(* Logix 5000 project; controller Ceca_1650T_Press 5069-L306ERM rev 32.12; software revision 32.02; part 3 of 3 *)
(* tags used below, declared in another part *)
   AUTO_CYCLE_ENABLED : BOOL;   // M0014 HMI SELECTION
   AUTO_CYCLE_SELECTED : BOOL;   // HMI BUTTON/SELECTION B0102
   AUTO_CYCLE_STOP_PB : BOOL;   // B0024
   AUTO_ONE_CYCLE_ENABLED : BOOL;   // M0013 HMI SELECTION
   AUTO_ONE_CYCLE_SELECTED : BOOL;   // HMI BUTTON/SELECTION B0101
   AUTO_UPPER_ASSIST : BOOL;   // ENCODER SIGNAL B0152
   AUTO_UPPER_ASSIST_POSITION_MINUS : REAL;
   AUTO_UPPER_ASSIST_POSITION_PLUS : REAL;
   AUTO_UPPER_LIMIT : BOOL;   // ENCODER SIGNAL B0151
   AUTO_UPPER_LIMIT_POSITION_MINUS : REAL;
   AUTO_UPPER_LIMIT_POSITION_PLUS : REAL;
   BLANKING_OFF_SIGNAL : TIMER;   // T0018
   BLANKING_PS_ENABLED : BOOL;   // M0018
   BOLSTER_DISABLED : BOOL;   // M0010
   CYCLE_STOP : BOOL;   // M0246
   DIE_CHANGE_ENABLED : BOOL;   // M0015
   DIE_CHANGE_MODE : BOOL;   // HMI BUTTON/SELECTION B0103
   DIE_SET_CHANGING : BOOL;   // B0037
   DIE_SET_CYLINDER_IN_PB : BOOL;   // B0076
   DIE_SET_CYLINDER_OUT : BOOL;   // M0217
   DIE_SET_CYLINDER_OUT_PB : BOOL;   // B0077
   DRAW_UP_ASSIST : BOOL;   // M007C
   FILTER_CLOGGED_FAULT : BOOL;   // M0023
   FRONT_SUTTER_ON_LIMIT : BOOL;   // B000C
   HMI_START_PUMPS : BOOL;   // HMI BUTTON
   INCH_ENABLED : BOOL;   // M0012 HMI SELECTION
   INCHING_SELECTED : BOOL;   // HMI BUTTON/SELECTION B0100
   Job_Call_Recipe : Recipe_Setup[50];
   L_DIECUSHION_AUTO_UP_ASSIST : BOOL;   // ENCODER SIGNAL B015A
   L_DIECUSHION_AUTO_UP_LIMIT : BOOL;   // B0156 ENCODER SIGNAL
   load_PB : BOOL;
   LOCKING_OFF_ASSIST : BOOL;   // M0032
   LUBE_LEVEL_FAULT : BOOL;   // M0022
   Machine_Current_Job : DINT;
   MAIN_PRESS_DOWN : BOOL;   // M0045
   MAIN_PRESS_POSITION_SICK : REAL;
   MAIN_PRESS_SLOW_DOWN : BOOL;   // M0046
   MAIN_PRESS_SLOW_UP : BOOL;   // M0042
   MAIN_PRESS_UP : BOOL;   // M0041
   MAIN_UPPER_LIMIT : BOOL;   // B0000
   OIL_COOLER_START : BOOL;   // B0144
   OIL_TEMP_TOO_HIGH : BOOL;   // B0143
   OIL_TEMP_WARM_UP_ON_SELECT : BOOL;   // B002C HMI BUTTON
   OIL_TEMP_WARM_UP_START : BOOL;   // B0038
   OIL_TEMPERATURE_FAULT : BOOL;   // M0025
   OIL_WORKING_LEVEL_FAULT : BOOL;   // M0021
   OPERATION_ON : BOOL;   // B0020
   PILOT_CHECK_OPEN_VALVE : BOOL;   // B0048
   PILOT_PUMP_HIGH_PRESSURE_VALVE : BOOL;   // B0060
   PILOT_PUMP_MIDDLE_PRESSURE_VALVE : BOOL;   // B0062
   PILOT_PUMP_ON : BOOL;   // B002E
   PRESS_AUTO_RUN : BOOL;   // M0069
   PRESS_HAS_A_FAULT : BOOL;   // M0027
   PRESS_HAS_A_FAULT_2 : BOOL;   // M0028
   PUMP_RUN : BOOL;   // B0021
   PUMP_START : BOOL;   // B1000
   PUMP_STOP_SIGNAL : BOOL;   // B0030
   R_DIECUSHION_AUTO_UP_ASSIST : BOOL;   // B015B ENCODER SIGNAL
   R_DIECUSHION_AUTO_UP_LIMIT : BOOL;   // B0158 ENCODER SIGNAL
   REAR_SHUTTER_ON_LIMIT : BOOL;   // B000D
   Recipe_Max : DINT;
   Recipe_Name_Pointer : DINT;
   Recipe_Number : COUNTER;
   Save_Delay : TIMER;
   save_pb : BOOL;
   Scroll_Down : BOOL;
   Scroll_up : BOOL;
   SickAFxWS_Enc1_AOI : SICK_AFX60_A101WS_A103WS_AOI;
   SickAFxWS_Enc1_Cyclic_GetSet : BOOL;
   SickAFxWS_Enc1_Init_GetSet : BOOL;
   SickAFxWS_Enc1_Timer_GetSet : TIMER;
   SLIDE_SLOW_DOWN_SIGNAL : BOOL;   // B0154 ENCODER SIGNAL
   SLIDE_SLOW_DOWN_SIGNAL_POSITION_MINUS : REAL;
   SLIDE_SLOW_DOWN_SIGNAL_POSITION_PLUS : REAL;
   TRM1 : BOOL;   // B1003
   TRM1_TIMER : TIMER;   // 5 SECONDS
   TRM2 : BOOL;   // B1001
   TRM2_TIMER : TIMER;   // 5 SECONDS
   TRM3 : BOOL;   // B1002
   TRM3_TIMER : TIMER;   // 1 SECOND
   WARM_UP_FINISHED : BOOL;   // M009E
   WARM_UP_OFF_TEMP : BOOL;   // B0027
   WARM_UP_ON : BOOL;   // M009D
   WARM_UP_ON_TIMING : TIMER;   // T0023
   WARM_UP_SELECT_OFF_TIMER : TIMER;   // T0024
   WARM_UP_SELECT_ON_TIMER : TIMER;   // T0025
(* MainProgram, continued *)

ROUTINE Modes   (* ladder *)
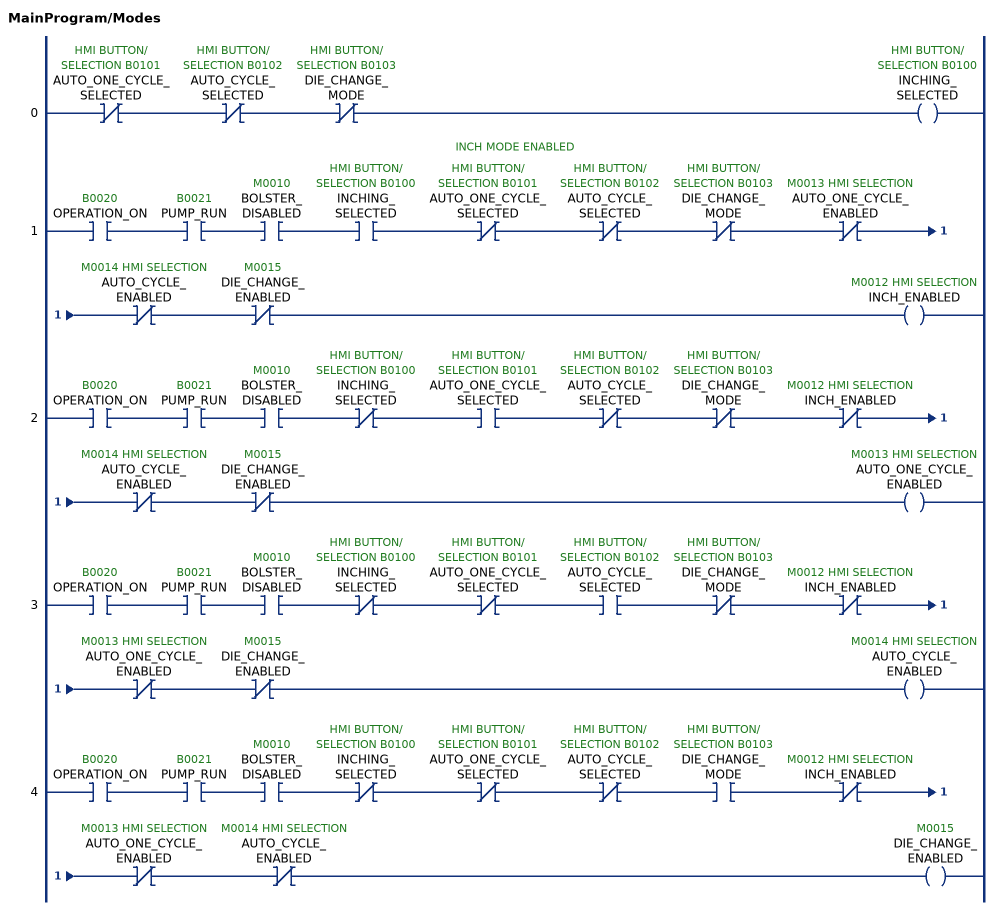
   0: XIO(AUTO_ONE_CYCLE_SELECTED)XIO(AUTO_CYCLE_SELECTED)XIO(DIE_CHANGE_MODE)OTE(INCHING_SELECTED);
   // INCH MODE ENABLED
   1: XIC(OPERATION_ON)XIC(PUMP_RUN)XIC(BOLSTER_DISABLED)XIC(INCHING_SELECTED)XIO(AUTO_ONE_CYCLE_SELECTED)XIO(AUTO_CYCLE_SELECTED)XIO(DIE_CHANGE_MODE)XIO(AUTO_ONE_CYCLE_ENABLED)XIO(AUTO_CYCLE_ENABLED)XIO(DIE_CHANGE_ENABLED)OTE(INCH_ENABLED);
   2: XIC(OPERATION_ON)XIC(PUMP_RUN)XIC(BOLSTER_DISABLED)XIO(INCHING_SELECTED)XIC(AUTO_ONE_CYCLE_SELECTED)XIO(AUTO_CYCLE_SELECTED)XIO(DIE_CHANGE_MODE)XIO(INCH_ENABLED)XIO(AUTO_CYCLE_ENABLED)XIO(DIE_CHANGE_ENABLED)OTE(AUTO_ONE_CYCLE_ENABLED);
   3: XIC(OPERATION_ON)XIC(PUMP_RUN)XIC(BOLSTER_DISABLED)XIO(INCHING_SELECTED)XIO(AUTO_ONE_CYCLE_SELECTED)XIC(AUTO_CYCLE_SELECTED)XIO(DIE_CHANGE_MODE)XIO(INCH_ENABLED)XIO(AUTO_ONE_CYCLE_ENABLED)XIO(DIE_CHANGE_ENABLED)OTE(AUTO_CYCLE_ENABLED);
   4: XIC(OPERATION_ON)XIC(PUMP_RUN)XIC(BOLSTER_DISABLED)XIO(INCHING_SELECTED)XIO(AUTO_ONE_CYCLE_SELECTED)XIO(AUTO_CYCLE_SELECTED)XIC(DIE_CHANGE_MODE)XIO(INCH_ENABLED)XIO(AUTO_ONE_CYCLE_ENABLED)XIO(AUTO_CYCLE_ENABLED)OTE(DIE_CHANGE_ENABLED);
END_ROUTINE

ROUTINE Outputs   (* ladder *)
END_ROUTINE

ROUTINE Pilot_Pump   (* ladder *)
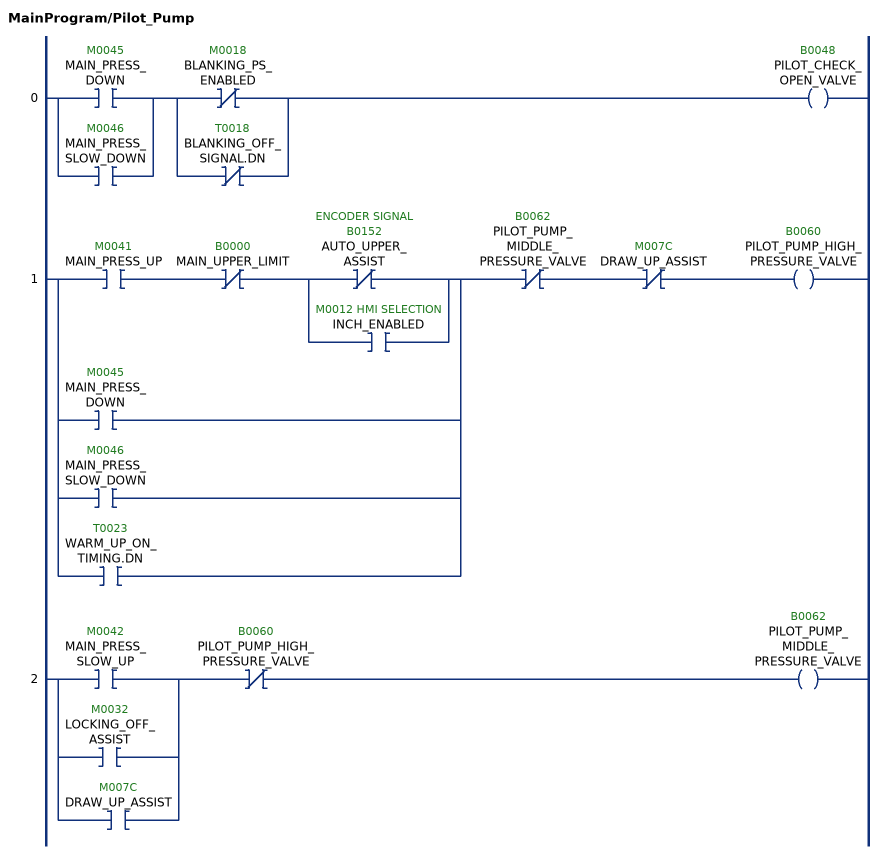
   0: [XIC(MAIN_PRESS_DOWN) ,XIC(MAIN_PRESS_SLOW_DOWN) ][XIO(BLANKING_PS_ENABLED) ,XIO(BLANKING_OFF_SIGNAL.DN) ]OTE(PILOT_CHECK_OPEN_VALVE);
   1: [XIC(MAIN_PRESS_UP) XIO(MAIN_UPPER_LIMIT) [XIO(AUTO_UPPER_ASSIST) ,XIC(INCH_ENABLED) ] ,XIC(MAIN_PRESS_DOWN) ,XIC(MAIN_PRESS_SLOW_DOWN) ,XIC(WARM_UP_ON_TIMING.DN) ]XIO(PILOT_PUMP_MIDDLE_PRESSURE_VALVE)XIO(DRAW_UP_ASSIST)OTE(PILOT_PUMP_HIGH_PRESSURE_VALVE);
   2: [XIC(MAIN_PRESS_SLOW_UP) ,XIC(LOCKING_OFF_ASSIST) ,XIC(DRAW_UP_ASSIST) ]XIO(PILOT_PUMP_HIGH_PRESSURE_VALVE)OTE(PILOT_PUMP_MIDDLE_PRESSURE_VALVE);
END_ROUTINE

ROUTINE Recipe   (* ladder *)
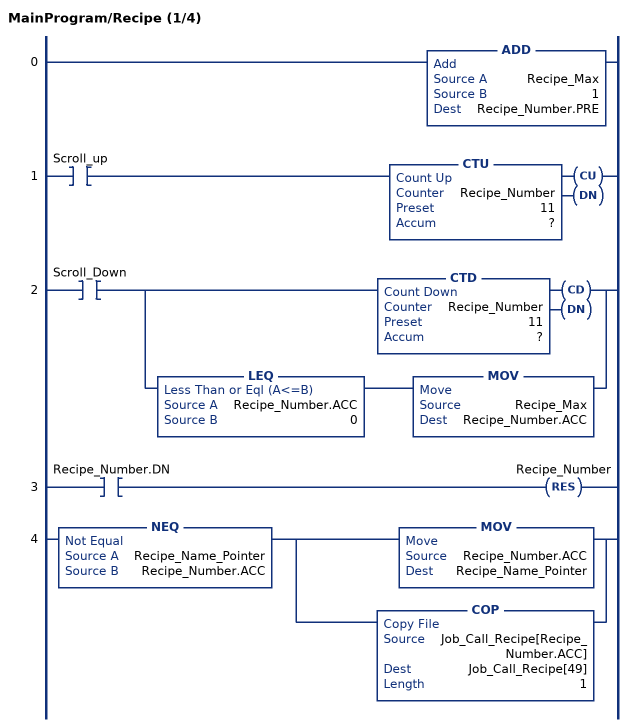
   0: ADD(Recipe_Max,1,Recipe_Number.PRE);
   1: XIC(Scroll_up)CTU(Recipe_Number,?,?);
   2: XIC(Scroll_Down)[CTD(Recipe_Number,?,?) ,LEQ(Recipe_Number.ACC,0) MOV(Recipe_Max,Recipe_Number.ACC) ];
   3: XIC(Recipe_Number.DN)RES(Recipe_Number);
   4: NEQ(Recipe_Name_Pointer,Recipe_Number.ACC)[MOV(Recipe_Number.ACC,Recipe_Name_Pointer) ,COP(Job_Call_Recipe[Recipe_Number.ACC],Job_Call_Recipe[49],1) ];
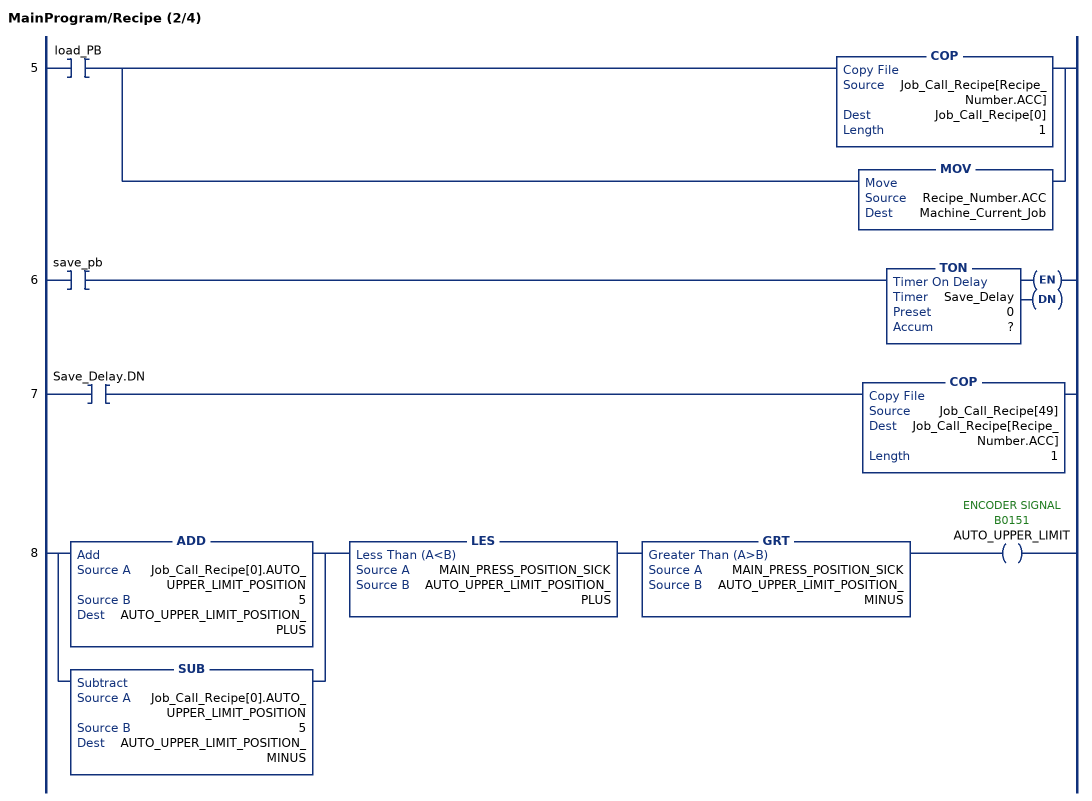
   5: XIC(load_PB)[COP(Job_Call_Recipe[Recipe_Number.ACC],Job_Call_Recipe[0],1) ,MOV(Recipe_Number.ACC,Machine_Current_Job) ];
   6: XIC(save_pb)TON(Save_Delay,?,?);
   7: XIC(Save_Delay.DN)COP(Job_Call_Recipe[49],Job_Call_Recipe[Recipe_Number.ACC],1);
   8: [ADD(Job_Call_Recipe[0].AUTO_UPPER_LIMIT_POSITION,5,AUTO_UPPER_LIMIT_POSITION_PLUS) ,SUB(Job_Call_Recipe[0].AUTO_UPPER_LIMIT_POSITION,5,AUTO_UPPER_LIMIT_POSITION_MINUS) ]LES(MAIN_PRESS_POSITION_SICK,AUTO_UPPER_LIMIT_POSITION_PLUS)GRT(MAIN_PRESS_POSITION_SICK,AUTO_UPPER_LIMIT_POSITION_MINUS)OTE(AUTO_UPPER_LIMIT);
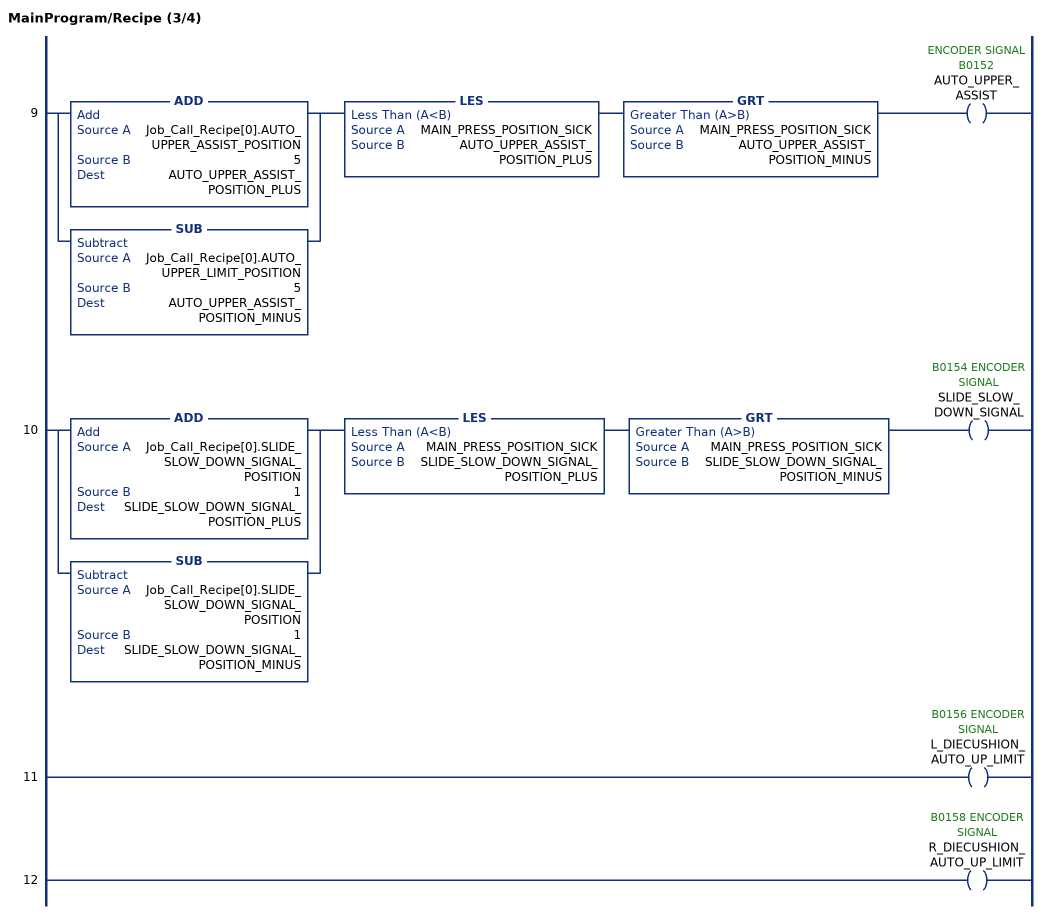
   9: [ADD(Job_Call_Recipe[0].AUTO_UPPER_ASSIST_POSITION,5,AUTO_UPPER_ASSIST_POSITION_PLUS) ,SUB(Job_Call_Recipe[0].AUTO_UPPER_LIMIT_POSITION,5,AUTO_UPPER_ASSIST_POSITION_MINUS) ]LES(MAIN_PRESS_POSITION_SICK,AUTO_UPPER_ASSIST_POSITION_PLUS)GRT(MAIN_PRESS_POSITION_SICK,AUTO_UPPER_ASSIST_POSITION_MINUS)OTE(AUTO_UPPER_ASSIST);
   10: [ADD(Job_Call_Recipe[0].SLIDE_SLOW_DOWN_SIGNAL_POSITION,1,SLIDE_SLOW_DOWN_SIGNAL_POSITION_PLUS) ,SUB(Job_Call_Recipe[0].SLIDE_SLOW_DOWN_SIGNAL_POSITION,1,SLIDE_SLOW_DOWN_SIGNAL_POSITION_MINUS) ]LES(MAIN_PRESS_POSITION_SICK,SLIDE_SLOW_DOWN_SIGNAL_POSITION_PLUS)GRT(MAIN_PRESS_POSITION_SICK,SLIDE_SLOW_DOWN_SIGNAL_POSITION_MINUS)OTE(SLIDE_SLOW_DOWN_SIGNAL);
   11: OTE(L_DIECUSHION_AUTO_UP_LIMIT);
   12: OTE(R_DIECUSHION_AUTO_UP_LIMIT);
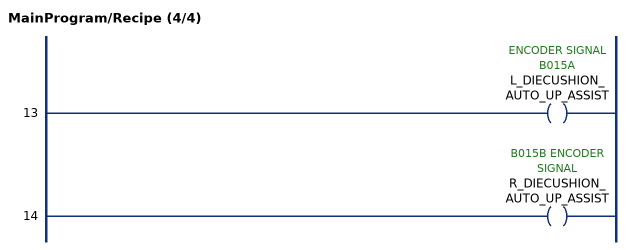
   13: OTE(L_DIECUSHION_AUTO_UP_ASSIST);
   14: OTE(R_DIECUSHION_AUTO_UP_ASSIST);
END_ROUTINE

ROUTINE Safety   (* ladder *)
END_ROUTINE

ROUTINE SickAFx_A101WS_A103WS_FB_Enc1_GetSet   (* ladder *)
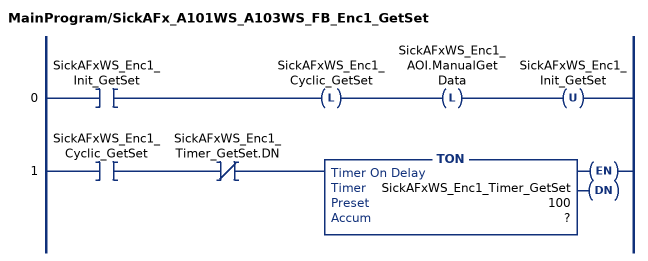
   0: XIC(SickAFxWS_Enc1_Init_GetSet)OTL(SickAFxWS_Enc1_Cyclic_GetSet)OTL(SickAFxWS_Enc1_AOI.ManualGetData)OTU(SickAFxWS_Enc1_Init_GetSet);
   1: XIC(SickAFxWS_Enc1_Cyclic_GetSet)XIO(SickAFxWS_Enc1_Timer_GetSet.DN)TON(SickAFxWS_Enc1_Timer_GetSet,?,?);
END_ROUTINE

ROUTINE Stop   (* ladder *)
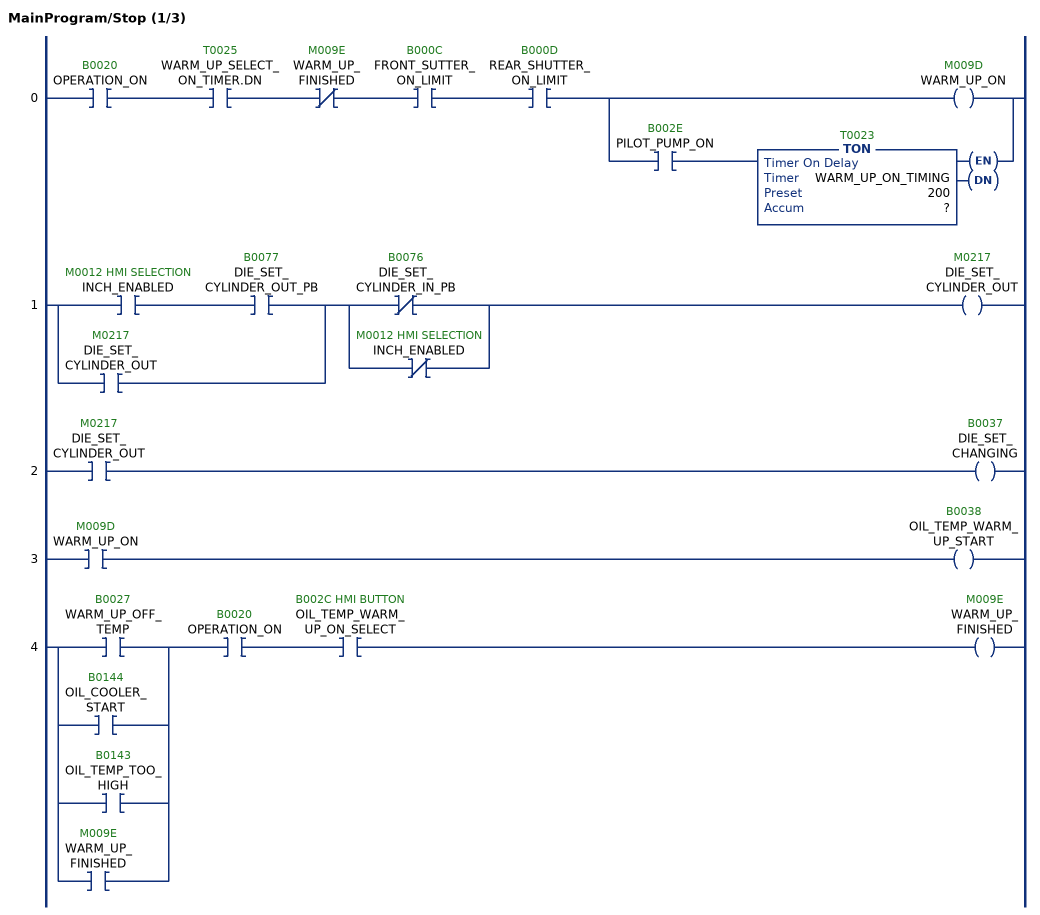
   0: XIC(OPERATION_ON)XIC(WARM_UP_SELECT_ON_TIMER.DN)XIO(WARM_UP_FINISHED)XIC(FRONT_SUTTER_ON_LIMIT)XIC(REAR_SHUTTER_ON_LIMIT)[OTE(WARM_UP_ON) ,XIC(PILOT_PUMP_ON) TON(WARM_UP_ON_TIMING,?,?) ];
   1: [XIC(INCH_ENABLED) XIC(DIE_SET_CYLINDER_OUT_PB) ,XIC(DIE_SET_CYLINDER_OUT) ][XIO(DIE_SET_CYLINDER_IN_PB) ,XIO(INCH_ENABLED) ]OTE(DIE_SET_CYLINDER_OUT);
   2: XIC(DIE_SET_CYLINDER_OUT)OTE(DIE_SET_CHANGING);
   3: XIC(WARM_UP_ON)OTE(OIL_TEMP_WARM_UP_START);
   4: [XIC(WARM_UP_OFF_TEMP) ,XIC(OIL_COOLER_START) ,XIC(OIL_TEMP_TOO_HIGH) ,XIC(WARM_UP_FINISHED) ]XIC(OPERATION_ON)XIC(OIL_TEMP_WARM_UP_ON_SELECT)OTE(WARM_UP_FINISHED);
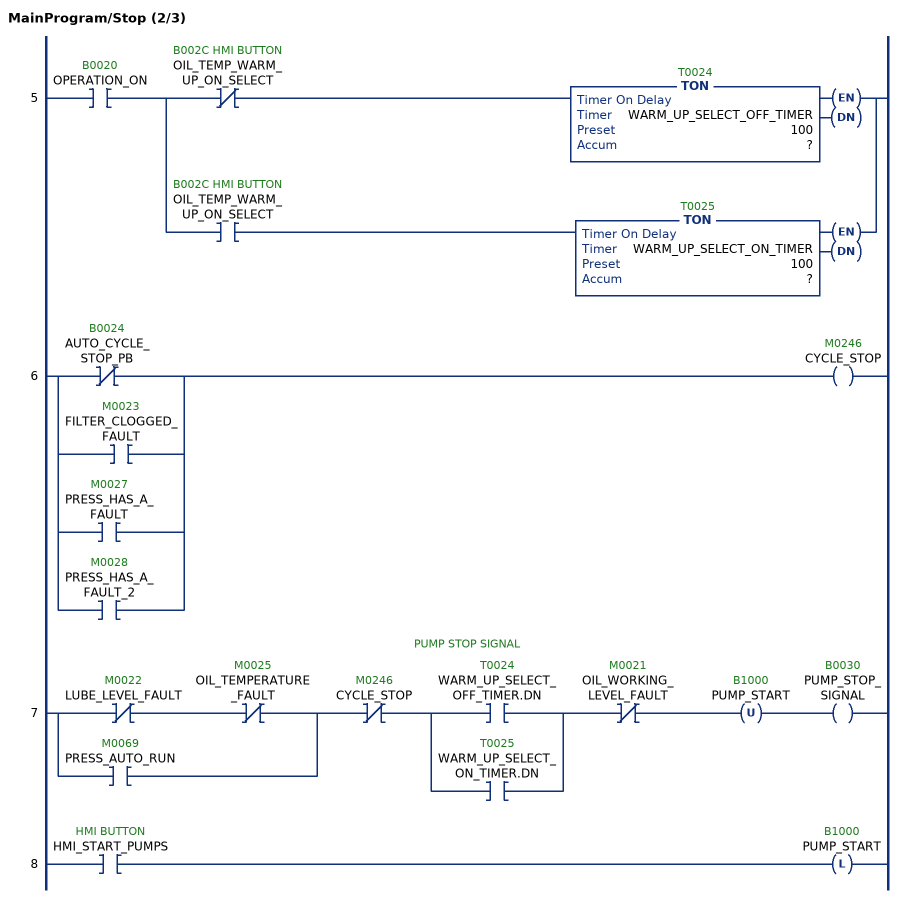
   5: XIC(OPERATION_ON)[XIO(OIL_TEMP_WARM_UP_ON_SELECT) TON(WARM_UP_SELECT_OFF_TIMER,?,?) ,XIC(OIL_TEMP_WARM_UP_ON_SELECT) TON(WARM_UP_SELECT_ON_TIMER,?,?) ];
   6: [XIO(AUTO_CYCLE_STOP_PB) ,XIC(FILTER_CLOGGED_FAULT) ,XIC(PRESS_HAS_A_FAULT) ,XIC(PRESS_HAS_A_FAULT_2) ]OTE(CYCLE_STOP);
   // PUMP STOP SIGNAL
   7: [XIO(LUBE_LEVEL_FAULT) XIO(OIL_TEMPERATURE_FAULT) ,XIC(PRESS_AUTO_RUN) ]XIO(CYCLE_STOP)[XIC(WARM_UP_SELECT_OFF_TIMER.DN) ,XIC(WARM_UP_SELECT_ON_TIMER.DN) ]XIO(OIL_WORKING_LEVEL_FAULT)OTU(PUMP_START)OTE(PUMP_STOP_SIGNAL);
   8: XIC(HMI_START_PUMPS)OTL(PUMP_START);
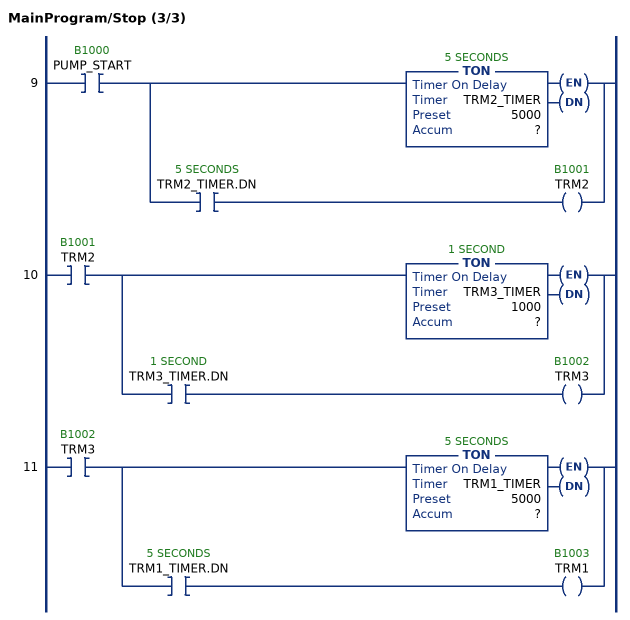
   9: XIC(PUMP_START)[TON(TRM2_TIMER,?,?) ,XIC(TRM2_TIMER.DN) OTE(TRM2) ];
   10: XIC(TRM2)[TON(TRM3_TIMER,?,?) ,XIC(TRM3_TIMER.DN) OTE(TRM3) ];
   11: XIC(TRM3)[TON(TRM1_TIMER,?,?) ,XIC(TRM1_TIMER.DN) OTE(TRM1) ];
END_ROUTINE
END_PROGRAM
